# EPICS autosave request: iocBoot/ioc13lab_linux/Galil_positions.req
file "CARS_32_motor_positions.req", P=$(P)
